ABB RobotStudio station: Solution_1_Template.rspag

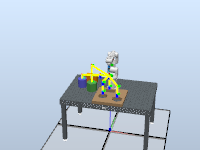
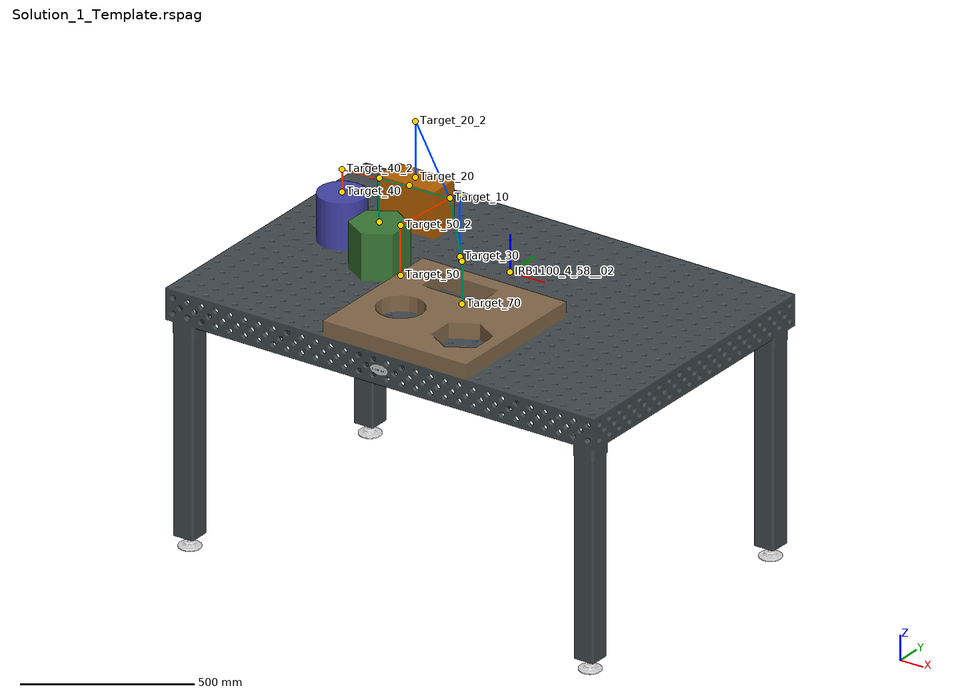
[picture v1: parts stored in the station drawn from their meshes, with robot base, taught points and paths (robot models come from the ABB library and are not in the file)]
--- station ---
Station Solution_1_Tutorial (saved by RobotStudio 21.4.9700.0)
Controller Controller1, task T_ROB1: task frame (RAPID world) sits at (0, 150, 830) mm, rotated rx 0 ry 0 rz -90 deg in the station
Controller Controller1
  mechanical unit ROB_1: IRB1100_4_58__02, 6 joints, base frame (0, 0, 0) mm
Layout (positions relative to the parent item):
  - table [part] at (-200, -500, 830) mm, size 500 x 500 x 50 mm
  - object_1 [part] at (-600, -150, 830) mm, size 200 x 100 x 150 mm
  - object_2 [part] at (-650, -150, 830) mm, size 149.5 x 149.7 x 150 mm
  - object_3 [part] at (-700, -200, 830) mm, size 155.5 x 179.5 x 150 mm
  - siegmund_1500_1000 [part], size 1500 x 1010.3 x 830 mm
  - object_11 [part] at (-200, -500, 830) mm, size 200 x 100 x 150 mm
  - object_22 [part] at (-200, -500, 830) mm, size 149.5 x 149.7 x 150 mm
  - object_33 [part] at (-200, -500, 830) mm, size 155.5 x 179.5 x 150 mm
  - IRB1100_4_58__02 [mechanism, from Robots\IRB1100_4_58__02.rslib] at (0, 150, 830) mm, rotated rx 0 ry 0 rz -90 deg; joint values [0, 0, 0, 0, 1.5708, 0] (rad or m)
  - smc_gripper [mechanism, from studio_home\smc_gripper.rslib] at (0, -150, 1383) mm, rotated rx 180 ry 0 rz 90 deg
  - Positioner_obj1 [smart component, from Components\Positioner.rslib]
      properties: Object=object_1; Position=[-0.6 -0.15 0.83]; Orientation=[0 0 0]; Reference=Global; ReferenceObject=(none)
  - Positioner_obj2 [smart component, from Components\Positioner.rslib]
      properties: Object=object_2; Position=[-0.65 -0.15 0.83]; Orientation=[0 0 0]; Reference=Global; ReferenceObject=(none)
  - Positioner_obj3 [smart component, from Components\Positioner.rslib]
      properties: Object=object_3; Position=[-0.7 -0.2 0.83]; Orientation=[0 0 0]; Reference=Global; ReferenceObject=(none)
  - Attacher_obj1 [smart component, from Components\Attacher.rslib]
      properties: Parent=smc_gripper; Flange=0; Child=object_1; Mount=false; Offset=[0 0 0]; Orientation=[0 0 0]
  - Detacher_obj1 [smart component, from Components\Detacher.rslib]
      properties: Child=object_1; KeepPosition=true
  - Detacher_obj2 [smart component, from Components\Detacher.rslib]
      properties: Child=object_2; KeepPosition=true
  - Detacher_obj3 [smart component, from Components\Detacher.rslib]
      properties: Child=object_3; KeepPosition=true
  - Attacher_obj2 [smart component, from Components\Attacher.rslib]
      properties: Parent=smc_gripper; Flange=0; Child=object_2; Mount=false; Offset=[0 0 0]; Orientation=[0 0 0]
  - Attacher_obj3 [smart component, from Components\Attacher.rslib]
      properties: Parent=smc_gripper; Flange=0; Child=object_3; Mount=false; Offset=[0 0 0]; Orientation=[0 0 0]
Attachment: smc_gripper is attached to IRB1100_4_58__02 / Link6
Station signals: DI obj1_home, DI obj2_home, DI obj3_home
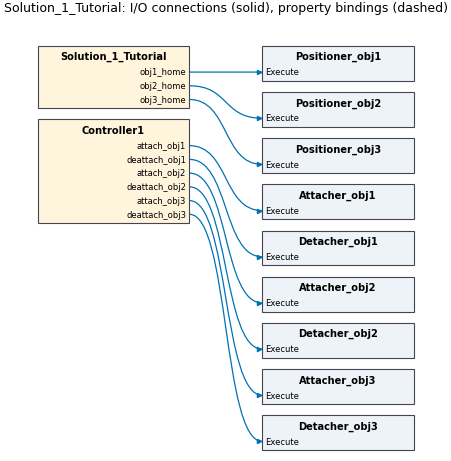
Station logic (signal -> signal, property => property):
  Solution_1_Tutorial.obj1_home -> Positioner_obj1.Execute
  Solution_1_Tutorial.obj2_home -> Positioner_obj2.Execute
  Solution_1_Tutorial.obj3_home -> Positioner_obj3.Execute
  Controller1.attach_obj1 -> Attacher_obj1.Execute
  Controller1.deattach_obj1 -> Detacher_obj1.Execute
  Controller1.attach_obj2 -> Attacher_obj2.Execute
  Controller1.deattach_obj2 -> Detacher_obj2.Execute
  Controller1.attach_obj3 -> Attacher_obj3.Execute
  Controller1.deattach_obj3 -> Detacher_obj3.Execute

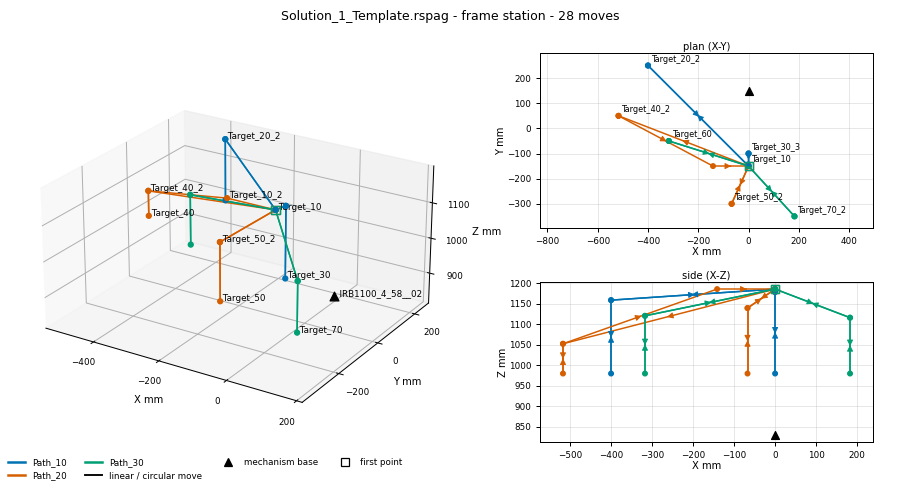
[picture p0: tool path of Solution_1_Template.rspag in frame station, 28 of 28 moves have a stored position in this frame; points joined in program order, loops and branches not executed]
--- Backups/Controller1/RAPID/TASK1/PROGMOD/CalibData.modx ---
MODULE CalibData
    PERS tooldata smc_gripper:=[TRUE,[[0,0.004,197.001],[1,0,0,0]],[1,[0.207,-0.496,71.18],[1,0,0,0],0,0,0]];
ENDMODULE

--- Backups/Controller1/RAPID/TASK1/PROGMOD/Module1.modx ---
MODULE Module1
        CONST robtarget Target_10:=[[300,0.004,355.999],[0,0,1,0],[0,0,0,0],[9E+09,9E+09,9E+09,9E+09,9E+09,9E+09]];
    CONST robtarget Target_20_2:=[[-100,-400,329.00332918],[0,0,1,0],[-2,0,-2,0],[9E+09,9E+09,9E+09,9E+09,9E+09,9E+09]];
    CONST robtarget Target_20:=[[-100,-400,150],[0,0,1,0],[-2,0,-2,0],[9E+09,9E+09,9E+09,9E+09,9E+09,9E+09]];
    CONST robtarget Target_30_3:=[[250,0,348.719268927],[0,0,1,0],[-1,0,-1,0],[9E+09,9E+09,9E+09,9E+09,9E+09,9E+09]];
    CONST robtarget Target_30:=[[250,0,150],[0,0,1,0],[-1,0,-1,0],[9E+09,9E+09,9E+09,9E+09,9E+09,9E+09]];
    CONST robtarget Target_40_2:=[[100,-517.298,222.628306773],[0,0,1,0],[0,0,0,0],[9E+09,9E+09,9E+09,9E+09,9E+09,9E+09]];
    CONST robtarget Target_40:=[[100,-517.298,150],[0,0,1,0],[0,0,0,0],[9E+09,9E+09,9E+09,9E+09,9E+09,9E+09]];
    CONST robtarget Target_10_2:=[[300,-141.413333438,355.999],[0,0,1,0],[-1,0,-1,0],[9E+09,9E+09,9E+09,9E+09,9E+09,9E+09]];
    CONST robtarget Target_50_2:=[[450,-67.298,309.693426029],[0,0,1,0],[0,0,0,0],[9E+09,9E+09,9E+09,9E+09,9E+09,9E+09]];
    CONST robtarget Target_50:=[[450,-67.298,150],[0,0,1,0],[0,0,0,0],[9E+09,9E+09,9E+09,9E+09,9E+09,9E+09]];
    CONST robtarget Target_60:=[[200,-317.298,290.802693742],[0,0,1,0],[0,0,0,0],[9E+09,9E+09,9E+09,9E+09,9E+09,9E+09]];
    CONST robtarget Target_60_2:=[[200,-317.298,150],[0,0,1,0],[0,0,0,0],[9E+09,9E+09,9E+09,9E+09,9E+09,9E+09]];
    CONST robtarget Target_70_2:=[[500,182.702,286.290213209],[0,0,1,0],[0,0,0,0],[9E+09,9E+09,9E+09,9E+09,9E+09,9E+09]];
    CONST robtarget Target_70:=[[500,182.702,150],[0,0,1,0],[0,0,0,0],[9E+09,9E+09,9E+09,9E+09,9E+09,9E+09]];

    PROC main()
        Path_10;
        Path_30;
        Path_20;
    ENDPROC
    PROC Path_10()
        MoveL Target_10,v100,z100,smc_gripper\WObj:=wobj0;
        !pick
        MoveL Target_20_2,v100,fine,smc_gripper\WObj:=wobj0;
        MoveL Target_20,v100,fine,smc_gripper\WObj:=wobj0;
        WaitTime 0.1;
        PulseDO attach_obj1;
        WaitTime 0.1;
        MoveL Target_20_2,v100,fine,smc_gripper\WObj:=wobj0;

        MoveL Target_10,v100,z100,smc_gripper\WObj:=wobj0;
        !place
        MoveL Target_30_3,v100,fine,smc_gripper\WObj:=wobj0;
        MoveL Target_30,v100,fine,smc_gripper\WObj:=wobj0;
        WaitTime 0.1;
        PulseDO deattach_obj1;
        WaitTime 0.1;
        MoveL Target_30_3,v100,fine,smc_gripper\WObj:=wobj0;

        MoveL Target_10,v100,z100,smc_gripper\WObj:=wobj0;
    ENDPROC
    PROC Path_20()
        MoveL Target_10,v100,fine,smc_gripper\WObj:=wobj0;
        !pick
        MoveL Target_40_2,v100,fine,smc_gripper\WObj:=wobj0;
        MoveL Target_40,v100,fine,smc_gripper\WObj:=wobj0;
        PulseDO attach_obj2;
        MoveL Target_40_2,v100,fine,smc_gripper\WObj:=wobj0;

        MoveL Target_10_2,v100,fine,smc_gripper\WObj:=wobj0;
        MoveL Target_10,v100,fine,smc_gripper\WObj:=wobj0;
        !place
        MoveL Target_50_2,v100,fine,smc_gripper\WObj:=wobj0;
        MoveL Target_50,v100,fine,smc_gripper\WObj:=wobj0;
        WaitTime 0.1;
        PulseDO deattach_obj2;
        WaitTime 0.1;
        MoveL Target_50_2,v100,fine,smc_gripper\WObj:=wobj0;

        MoveL Target_10,v100,fine,smc_gripper\WObj:=wobj0;
    ENDPROC
    PROC Path_30()
        MoveL Target_10,v100,fine,smc_gripper\WObj:=wobj0;
        !pick
        MoveL Target_60,v100,fine,smc_gripper\WObj:=wobj0;
        MoveL Target_60_2,v100,fine,smc_gripper\WObj:=wobj0;
        WaitTime 0.1;
        PulseDO attach_obj3;
        WaitTime 0.1;
        MoveL Target_60,v100,fine,smc_gripper\WObj:=wobj0;

        MoveL Target_10,v100,fine,smc_gripper\WObj:=wobj0;
        !place
        MoveL Target_70_2,v100,fine,smc_gripper\WObj:=wobj0;
        MoveL Target_70,v100,fine,smc_gripper\WObj:=wobj0;
        WaitTime 0.1;
        PulseDO deattach_obj3;
        WaitTime 0.1;
        MoveL Target_70_2,v100,fine,smc_gripper\WObj:=wobj0;
        MoveL Target_10,v1000,z100,smc_gripper\WObj:=wobj0;
    ENDPROC
ENDMODULE

--- Backups/Controller1/SYSPAR/EIO.cfg ---
EIO:CFG_1.0:7:0::
#
EIO_SIGNAL:

      -Name "attach_obj1" -SignalType "DO"

      -Name "attach_obj2" -SignalType "DO"

      -Name "attach_obj3" -SignalType "DO"

      -Name "deattach_obj1" -SignalType "DO"

      -Name "deattach_obj2" -SignalType "DO"

      -Name "deattach_obj3" -SignalType "DO"

#CTRL_SIGNATURE:wFaTNvIl4adKNDjARSI58lNp9JBsUF4PdtDLc17vVf6Kzewnb0X8+gGsRX/MgEmwpwu9X5IrMnWDeERPEhSpIA==

--- Backups/Controller1/SYSPAR/PROC.cfg ---
PROC:CFG_1.0:7:0::

#CTRL_SIGNATURE:I+y2QaV15gWtHGM+5Z4idi3NiusZu29hLyokxM3ohwogLM8MfydOTWOtI2G6szFitByh5svEYsXD7agPogo+dQ==
